(* Logix 5000 project; controller R5_CSS vendor 1 type 14 code 74 rev 19.11; software revision 19.01; part 6 of 18 *)
(* tags used below, declared in another part *)
   AC102A : ANALYTICAL;   // QUENCH WATER CONDUCTIVITY CONTROL
   AlarmMaster : DINT;
   AlarmMasterDisable : BOOL;
   AlarmMasterResetTON : TIMER;
   AlarmResetPB : BOOL;
   FC101 : FLOW_CONTROL;   // QUENCH BASIN FLOW TRANSMITTER CONTROL
   FC108 : FLOW_CONTROL;   // QUENCH FEED FLOW TRANSMITTER
   FC140A : FLOW_CONTROL;   // QUENCH TOWER UPPER SPRAY FLOW CONTROL
   FC140B : FLOW_CONTROL;   // QUENCH TOWER LOWER SPRAY FLOW CONTROL
   FC365 : FLOW_CONTROL;   // COALESCER PROCESS IMPURITY FLOW CONTROL
   FireFlowAlarmFromUTL : BOOL;
   HMI_ShowReboot : BOOL;
   HMI_ShowRebootTmr : TIMER;
   Instrument_LOS : BOOL[32];
   LC205 : LEVEL_CONTROL;   // OVERHEAD CONDENSER BASIN LEVEL CONTROL
   LC302 : LEVEL_CONTROL;   // COALESCER OIL CHAMBER LEVEL CONTROL
   LC303A : LEVEL_CONTROL;   // AQUEOUS PHASE OF PRIMARY SETTLER
   Option_F1_Occupancy : BOOL;   // STATUS FROM UTL PLC 0=DISABLED 1=ENABLED
   P101_OK_TON : TIMER;
   P101A_OK : BOOL;
   P101B_OK : BOOL;
   P302A : PUMP_CONTROL;
   P302B : PUMP_CONTROL;
   P303_OK_TON : TIMER;
   P303A_OK : BOOL;
   P303B_OK : BOOL;
   PC101A : PRESSURE_CONTROL;   // LOWER QUENCH TOWER PRESSURE TRANSMITTER
   PC101B : PRESSURE_CONTROL;   // UPPER QUENCH TOWER PRESSURE TRANSMITTER PRESSURE CONTOL
   PC407B : PRESSURE_CONTROL;   // POST HX LOW PRESSURE TRANSMITTER
   TC101A : TEMP_CONTROL;   // QUENCH BASIN TRANSFER BASIN A TEMPERATURE CONTROL
   TC108 : TEMP_CONTROL;   // QUENCH TOWER EXIT GAS TEMPERATURE CONTROL
   TC114A : TEMP_CONTROL;   // QUENCH BASIN SHELL TEMPERATURE CONTROL
   TMR_FAULT : DINT;
   UTL_Comms : DINT[3];
   UTL_CommsLossAlm : BOOL;
(* MainProgram, continued *)

ROUTINE A4_Alarms_General   (* ladder *)
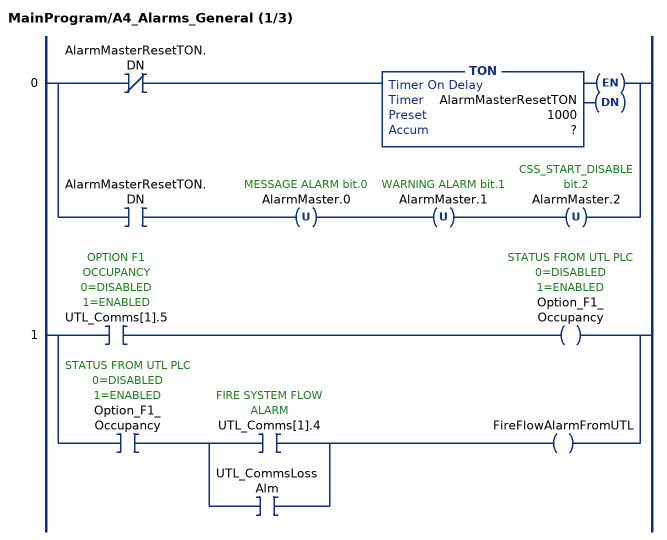
   0: [XIO(AlarmMasterResetTON.DN) TON(AlarmMasterResetTON,?,?) ,XIC(AlarmMasterResetTON.DN) OTU(AlarmMaster.0) OTU(AlarmMaster.1) OTU(AlarmMaster.2) ];
   1: [XIC(UTL_Comms[1].5) OTE(Option_F1_Occupancy) ,XIC(Option_F1_Occupancy) [XIC(UTL_Comms[1].4) ,XIC(UTL_CommsLossAlm) ] OTE(FireFlowAlarmFromUTL) ];
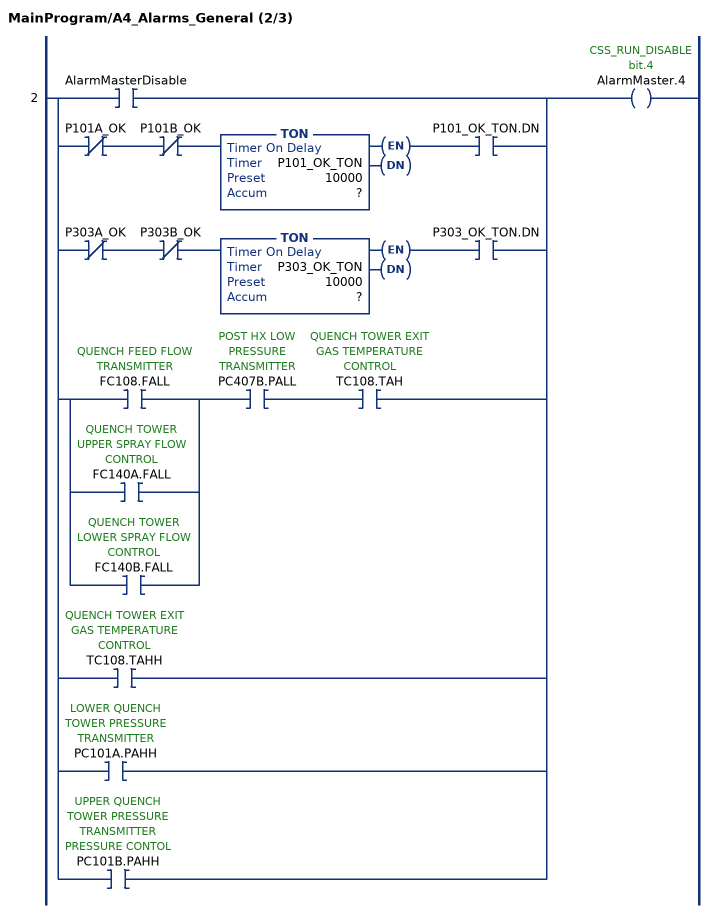
   2: [XIC(AlarmMasterDisable) ,XIO(P101A_OK) XIO(P101B_OK) TON(P101_OK_TON,?,?) XIC(P101_OK_TON.DN) ,XIO(P303A_OK) XIO(P303B_OK) TON(P303_OK_TON,?,?) XIC(P303_OK_TON.DN) ,[XIC(FC108.FALL) ,XIC(FC140A.FALL) ,XIC(FC140B.FALL) ] XIC(PC407B.PALL) XIC(TC108.TAH) ,XIC(TC108.TAHH) ,XIC(PC101A.PAHH) ,XIC(PC101B.PAHH) ]OTE(AlarmMaster.4);
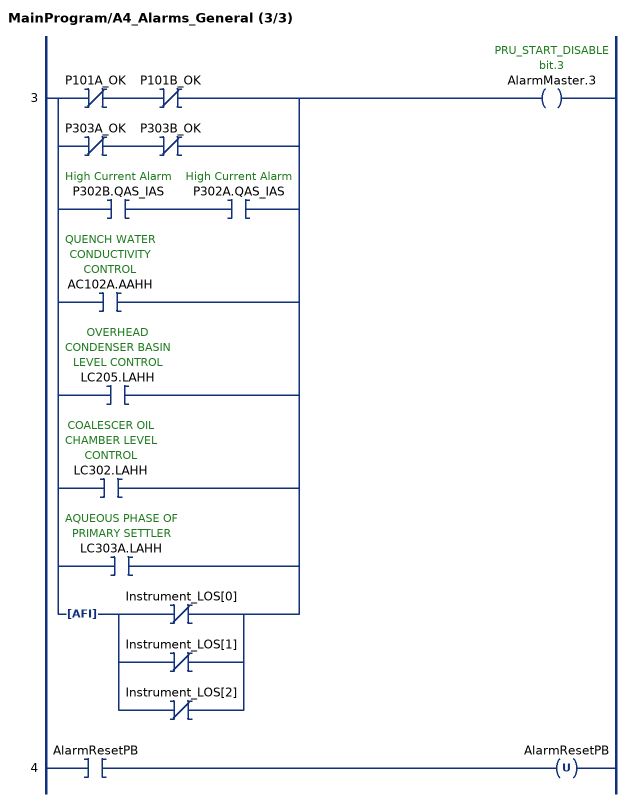
   3: [XIO(P101A_OK) XIO(P101B_OK) ,XIO(P303A_OK) XIO(P303B_OK) ,XIC(P302B.QAS_IAS) XIC(P302A.QAS_IAS) ,XIC(AC102A.AAHH) ,XIC(LC205.LAHH) ,XIC(LC302.LAHH) ,XIC(LC303A.LAHH) ,AFI() [XIO(Instrument_LOS[0]) ,XIO(Instrument_LOS[1]) ,XIO(Instrument_LOS[2]) ] ]OTE(AlarmMaster.3);
   4: XIC(AlarmResetPB)OTU(AlarmResetPB);
END_ROUTINE

ROUTINE A5a_LOAD_START_UP_PARAMETERS   (* ladder *)
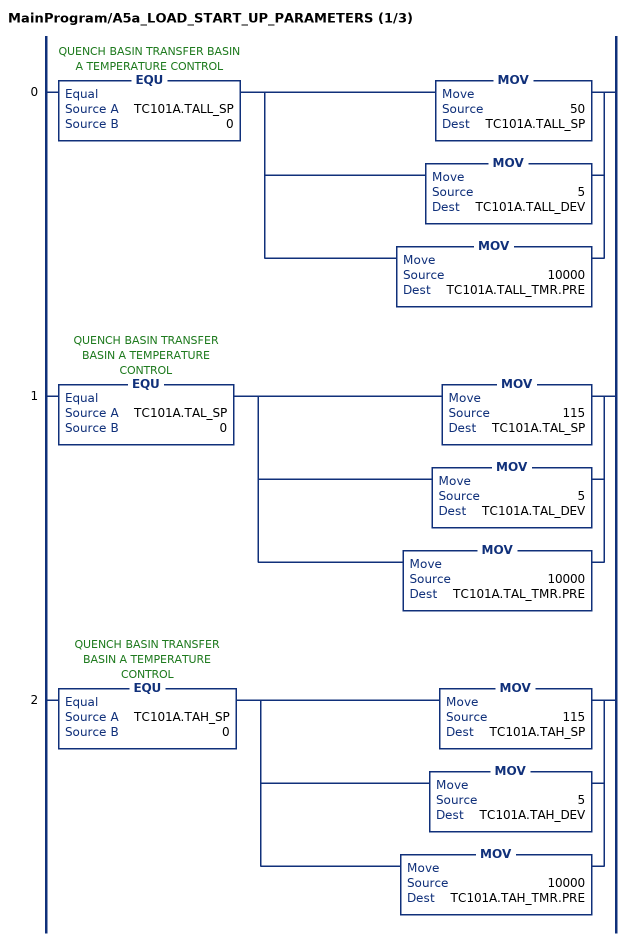
   0: EQU(TC101A.TALL_SP,0)[MOV(50,TC101A.TALL_SP) ,MOV(5,TC101A.TALL_DEV) ,MOV(10000,TC101A.TALL_TMR.PRE) ];
   1: EQU(TC101A.TAL_SP,0)[MOV(115,TC101A.TAL_SP) ,MOV(5,TC101A.TAL_DEV) ,MOV(10000,TC101A.TAL_TMR.PRE) ];
   2: EQU(TC101A.TAH_SP,0)[MOV(115,TC101A.TAH_SP) ,MOV(5,TC101A.TAH_DEV) ,MOV(10000,TC101A.TAH_TMR.PRE) ];
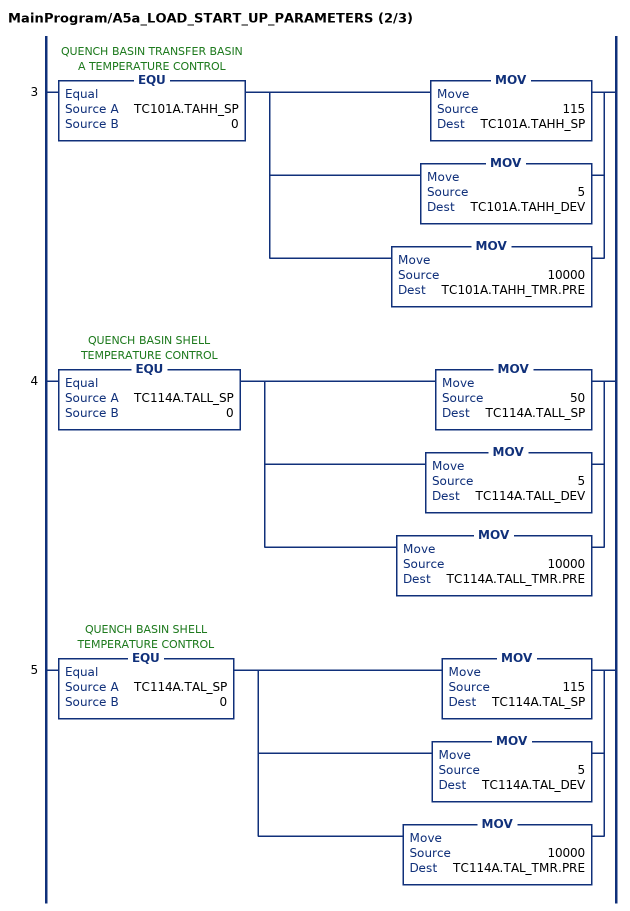
   3: EQU(TC101A.TAHH_SP,0)[MOV(115,TC101A.TAHH_SP) ,MOV(5,TC101A.TAHH_DEV) ,MOV(10000,TC101A.TAHH_TMR.PRE) ];
   4: EQU(TC114A.TALL_SP,0)[MOV(50,TC114A.TALL_SP) ,MOV(5,TC114A.TALL_DEV) ,MOV(10000,TC114A.TALL_TMR.PRE) ];
   5: EQU(TC114A.TAL_SP,0)[MOV(115,TC114A.TAL_SP) ,MOV(5,TC114A.TAL_DEV) ,MOV(10000,TC114A.TAL_TMR.PRE) ];
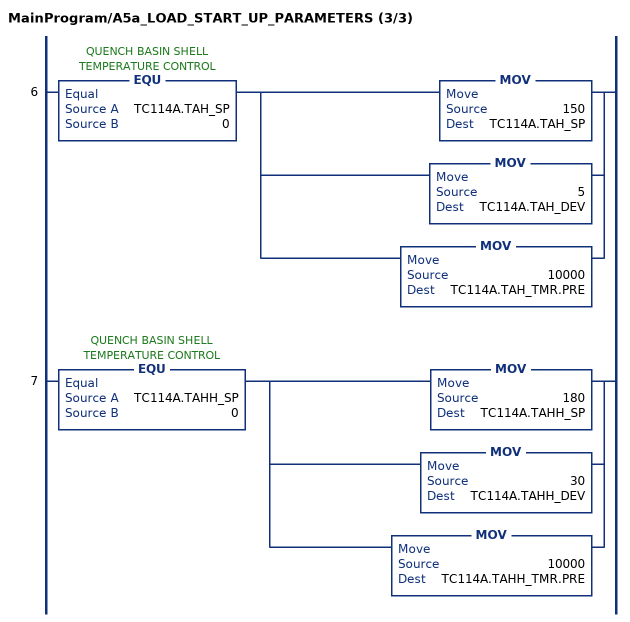
   6: EQU(TC114A.TAH_SP,0)[MOV(150,TC114A.TAH_SP) ,MOV(5,TC114A.TAH_DEV) ,MOV(10000,TC114A.TAH_TMR.PRE) ];
   7: EQU(TC114A.TAHH_SP,0)[MOV(180,TC114A.TAHH_SP) ,MOV(30,TC114A.TAHH_DEV) ,MOV(10000,TC114A.TAHH_TMR.PRE) ];
END_ROUTINE

ROUTINE A5b_LOCAL_HMI   (* ladder *)
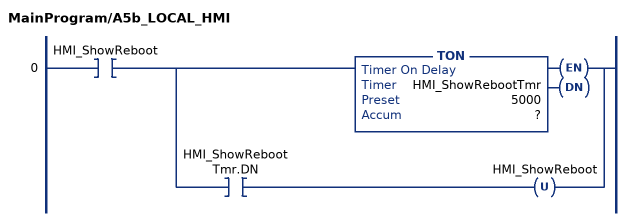
   0: XIC(HMI_ShowReboot)[TON(HMI_ShowRebootTmr,?,?) ,XIC(HMI_ShowRebootTmr.DN) OTU(HMI_ShowReboot) ];
END_ROUTINE

ROUTINE AT102A_QuenchWaterConductivity   (* ladder *)
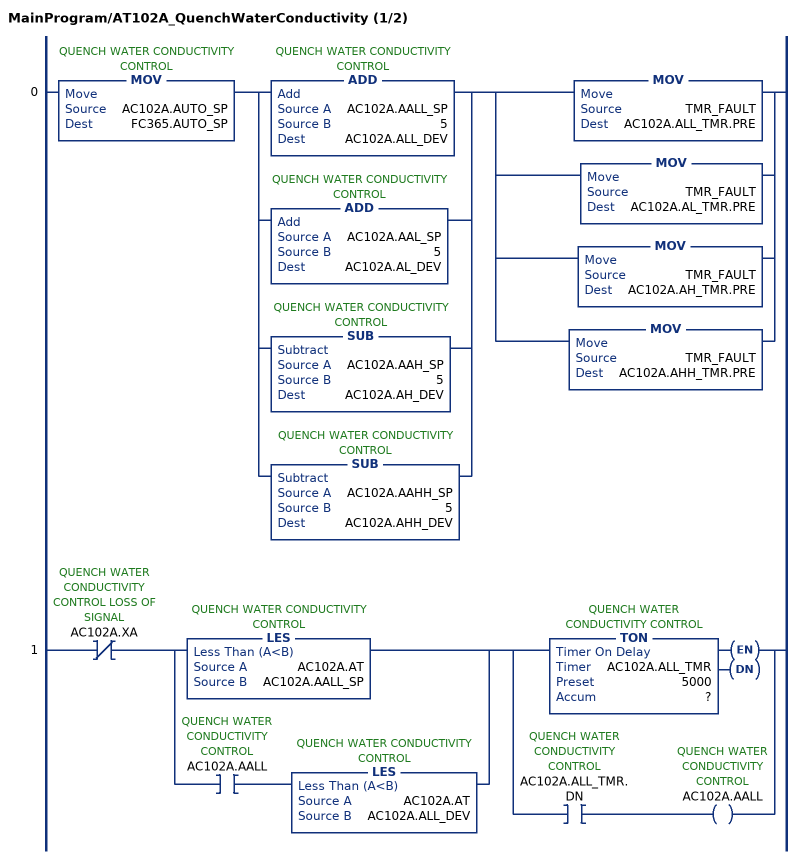
   0: MOV(AC102A.AUTO_SP,FC365.AUTO_SP)[ADD(AC102A.AALL_SP,5,AC102A.ALL_DEV) ,ADD(AC102A.AAL_SP,5,AC102A.AL_DEV) ,SUB(AC102A.AAH_SP,5,AC102A.AH_DEV) ,SUB(AC102A.AAHH_SP,5,AC102A.AHH_DEV) ][MOV(TMR_FAULT,AC102A.ALL_TMR.PRE) ,MOV(TMR_FAULT,AC102A.AL_TMR.PRE) ,MOV(TMR_FAULT,AC102A.AH_TMR.PRE) ,MOV(TMR_FAULT,AC102A.AHH_TMR.PRE) ];
   1: XIO(AC102A.XA)[LES(AC102A.AT,AC102A.AALL_SP) ,XIC(AC102A.AALL) LES(AC102A.AT,AC102A.ALL_DEV) ][TON(AC102A.ALL_TMR,?,?) ,XIC(AC102A.ALL_TMR.DN) OTE(AC102A.AALL) ];
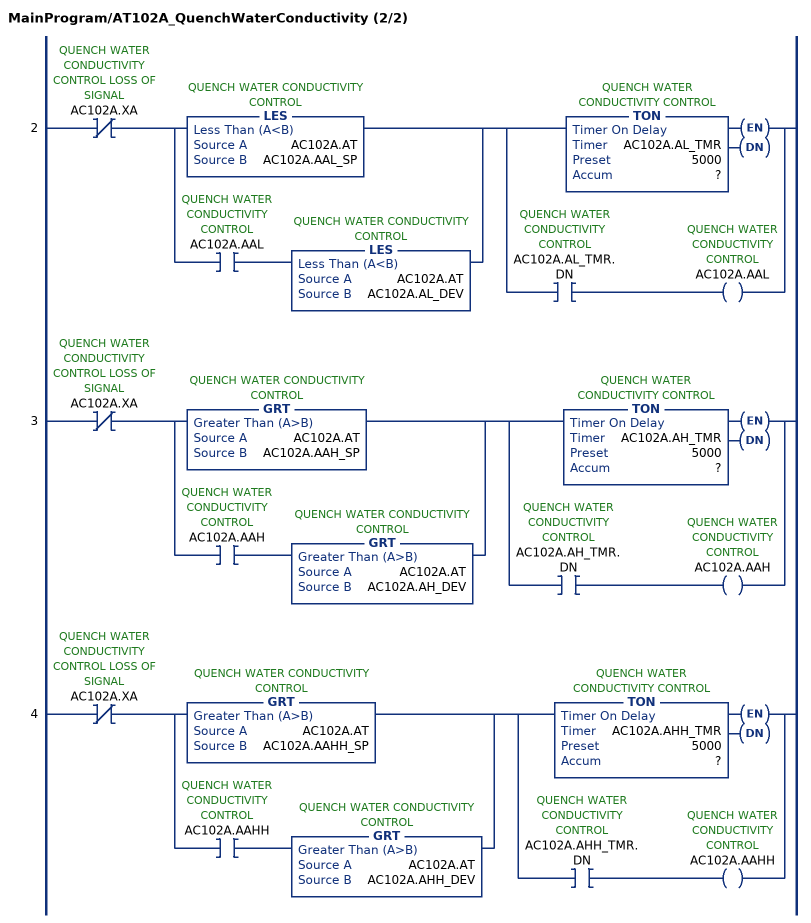
   2: XIO(AC102A.XA)[LES(AC102A.AT,AC102A.AAL_SP) ,XIC(AC102A.AAL) LES(AC102A.AT,AC102A.AL_DEV) ][TON(AC102A.AL_TMR,?,?) ,XIC(AC102A.AL_TMR.DN) OTE(AC102A.AAL) ];
   3: XIO(AC102A.XA)[GRT(AC102A.AT,AC102A.AAH_SP) ,XIC(AC102A.AAH) GRT(AC102A.AT,AC102A.AH_DEV) ][TON(AC102A.AH_TMR,?,?) ,XIC(AC102A.AH_TMR.DN) OTE(AC102A.AAH) ];
   4: XIO(AC102A.XA)[GRT(AC102A.AT,AC102A.AAHH_SP) ,XIC(AC102A.AAHH) GRT(AC102A.AT,AC102A.AHH_DEV) ][TON(AC102A.AHH_TMR,?,?) ,XIC(AC102A.AHH_TMR.DN) OTE(AC102A.AAHH) ];
END_ROUTINE

ROUTINE FC101_BasinFlow   (* ladder *)
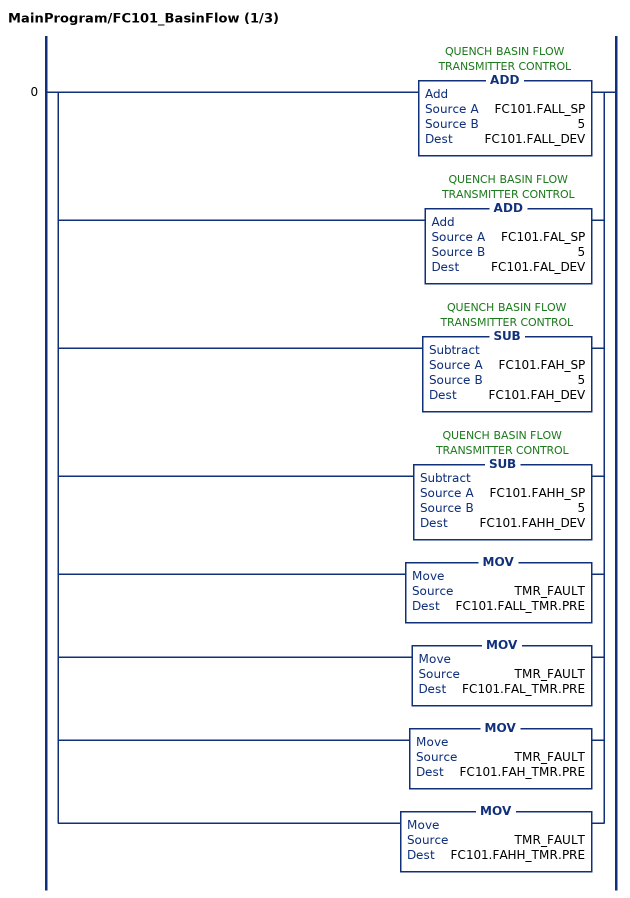
   0: [ADD(FC101.FALL_SP,5,FC101.FALL_DEV) ,ADD(FC101.FAL_SP,5,FC101.FAL_DEV) ,SUB(FC101.FAH_SP,5,FC101.FAH_DEV) ,SUB(FC101.FAHH_SP,5,FC101.FAHH_DEV) ,MOV(TMR_FAULT,FC101.FALL_TMR.PRE) ,MOV(TMR_FAULT,FC101.FAL_TMR.PRE) ,MOV(TMR_FAULT,FC101.FAH_TMR.PRE) ,MOV(TMR_FAULT,FC101.FAHH_TMR.PRE) ];
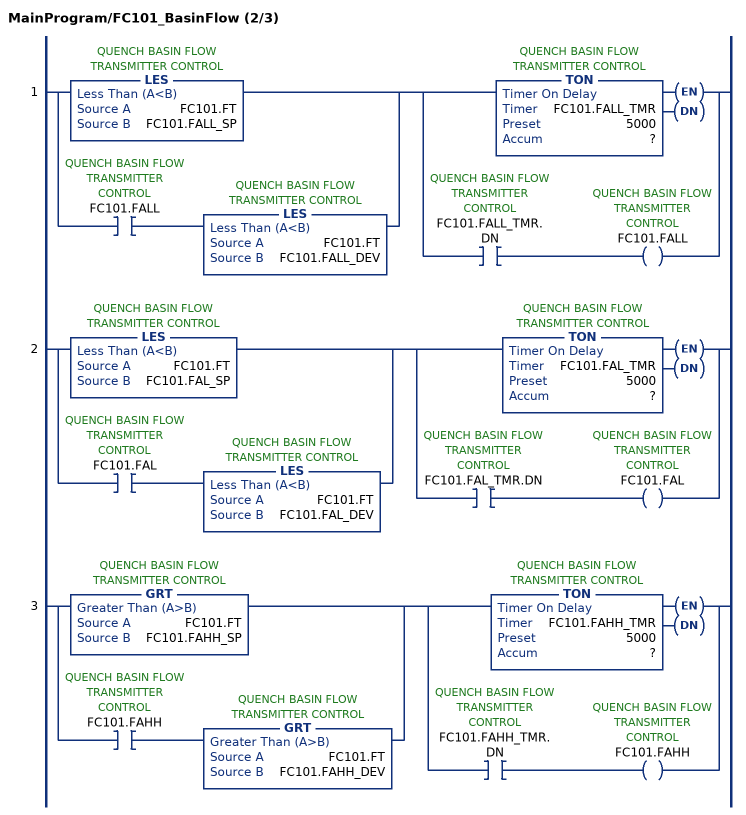
   1: [LES(FC101.FT,FC101.FALL_SP) ,XIC(FC101.FALL) LES(FC101.FT,FC101.FALL_DEV) ][TON(FC101.FALL_TMR,?,?) ,XIC(FC101.FALL_TMR.DN) OTE(FC101.FALL) ];
   2: [LES(FC101.FT,FC101.FAL_SP) ,XIC(FC101.FAL) LES(FC101.FT,FC101.FAL_DEV) ][TON(FC101.FAL_TMR,?,?) ,XIC(FC101.FAL_TMR.DN) OTE(FC101.FAL) ];
   3: [GRT(FC101.FT,FC101.FAHH_SP) ,XIC(FC101.FAHH) GRT(FC101.FT,FC101.FAHH_DEV) ][TON(FC101.FAHH_TMR,?,?) ,XIC(FC101.FAHH_TMR.DN) OTE(FC101.FAHH) ];
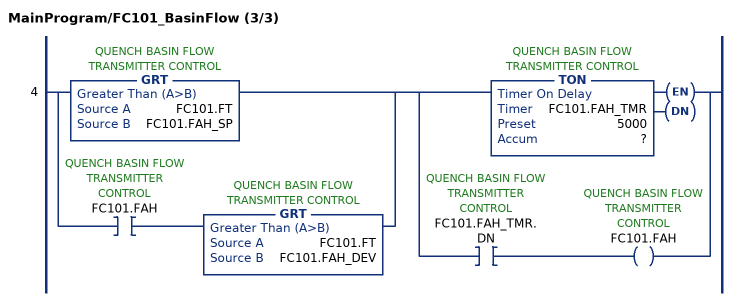
   4: [GRT(FC101.FT,FC101.FAH_SP) ,XIC(FC101.FAH) GRT(FC101.FT,FC101.FAH_DEV) ][TON(FC101.FAH_TMR,?,?) ,XIC(FC101.FAH_TMR.DN) OTE(FC101.FAH) ];
END_ROUTINE

ROUTINE FC108_QuenchTowerFlow   (* ladder *)
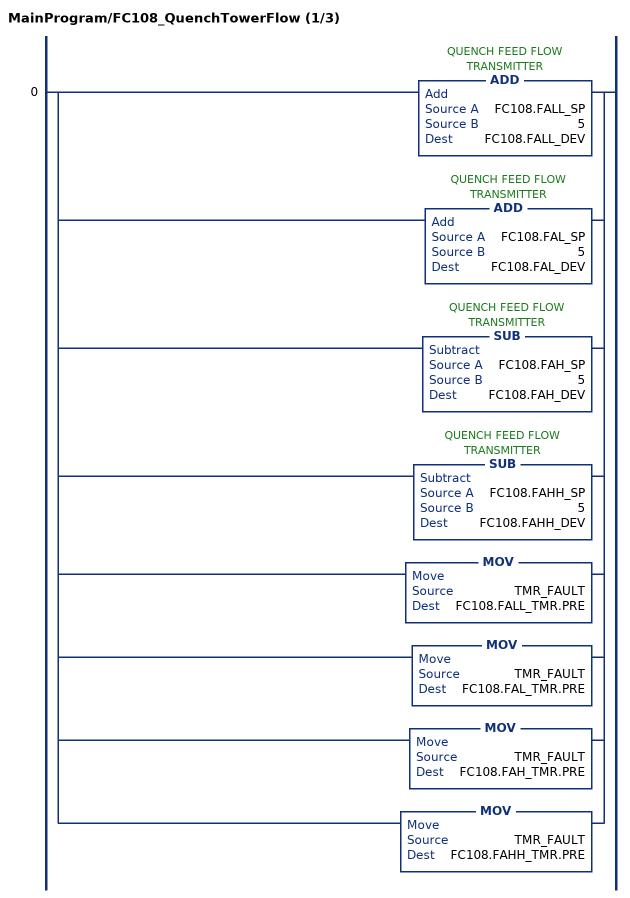
   0: [ADD(FC108.FALL_SP,5,FC108.FALL_DEV) ,ADD(FC108.FAL_SP,5,FC108.FAL_DEV) ,SUB(FC108.FAH_SP,5,FC108.FAH_DEV) ,SUB(FC108.FAHH_SP,5,FC108.FAHH_DEV) ,MOV(TMR_FAULT,FC108.FALL_TMR.PRE) ,MOV(TMR_FAULT,FC108.FAL_TMR.PRE) ,MOV(TMR_FAULT,FC108.FAH_TMR.PRE) ,MOV(TMR_FAULT,FC108.FAHH_TMR.PRE) ];
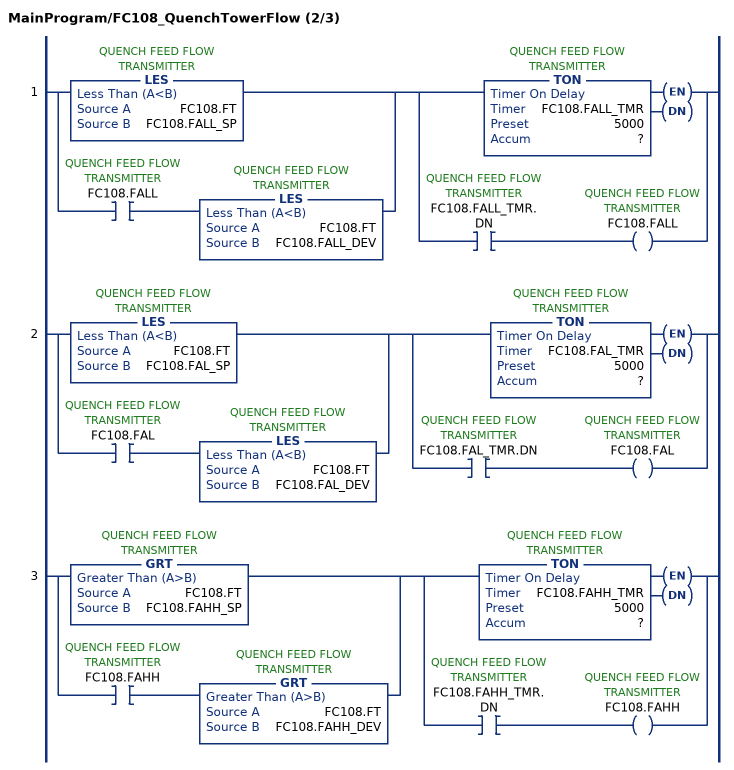
   1: [LES(FC108.FT,FC108.FALL_SP) ,XIC(FC108.FALL) LES(FC108.FT,FC108.FALL_DEV) ][TON(FC108.FALL_TMR,?,?) ,XIC(FC108.FALL_TMR.DN) OTE(FC108.FALL) ];
   2: [LES(FC108.FT,FC108.FAL_SP) ,XIC(FC108.FAL) LES(FC108.FT,FC108.FAL_DEV) ][TON(FC108.FAL_TMR,?,?) ,XIC(FC108.FAL_TMR.DN) OTE(FC108.FAL) ];
   3: [GRT(FC108.FT,FC108.FAHH_SP) ,XIC(FC108.FAHH) GRT(FC108.FT,FC108.FAHH_DEV) ][TON(FC108.FAHH_TMR,?,?) ,XIC(FC108.FAHH_TMR.DN) OTE(FC108.FAHH) ];
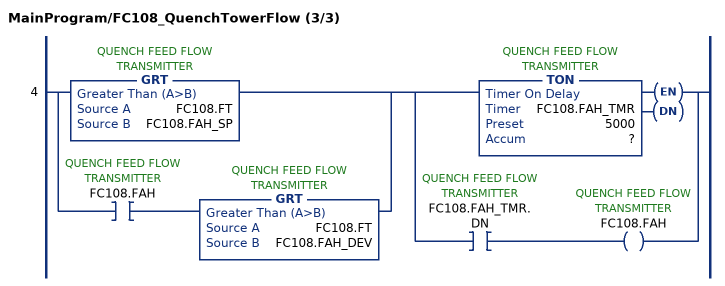
   4: [GRT(FC108.FT,FC108.FAH_SP) ,XIC(FC108.FAH) GRT(FC108.FT,FC108.FAH_DEV) ][TON(FC108.FAH_TMR,?,?) ,XIC(FC108.FAH_TMR.DN) OTE(FC108.FAH) ];
END_ROUTINE

ROUTINE FC140A_QuenchWaterUpperSprayFlow   (* ladder *)
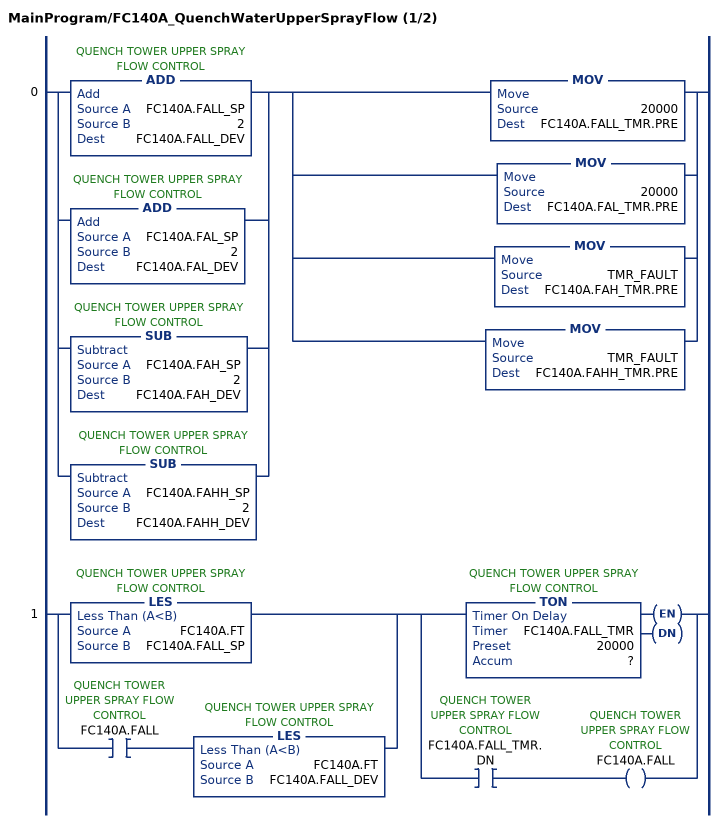
   0: [ADD(FC140A.FALL_SP,2,FC140A.FALL_DEV) ,ADD(FC140A.FAL_SP,2,FC140A.FAL_DEV) ,SUB(FC140A.FAH_SP,2,FC140A.FAH_DEV) ,SUB(FC140A.FAHH_SP,2,FC140A.FAHH_DEV) ][MOV(20000,FC140A.FALL_TMR.PRE) ,MOV(20000,FC140A.FAL_TMR.PRE) ,MOV(TMR_FAULT,FC140A.FAH_TMR.PRE) ,MOV(TMR_FAULT,FC140A.FAHH_TMR.PRE) ];
   1: [LES(FC140A.FT,FC140A.FALL_SP) ,XIC(FC140A.FALL) LES(FC140A.FT,FC140A.FALL_DEV) ][TON(FC140A.FALL_TMR,?,?) ,XIC(FC140A.FALL_TMR.DN) OTE(FC140A.FALL) ];
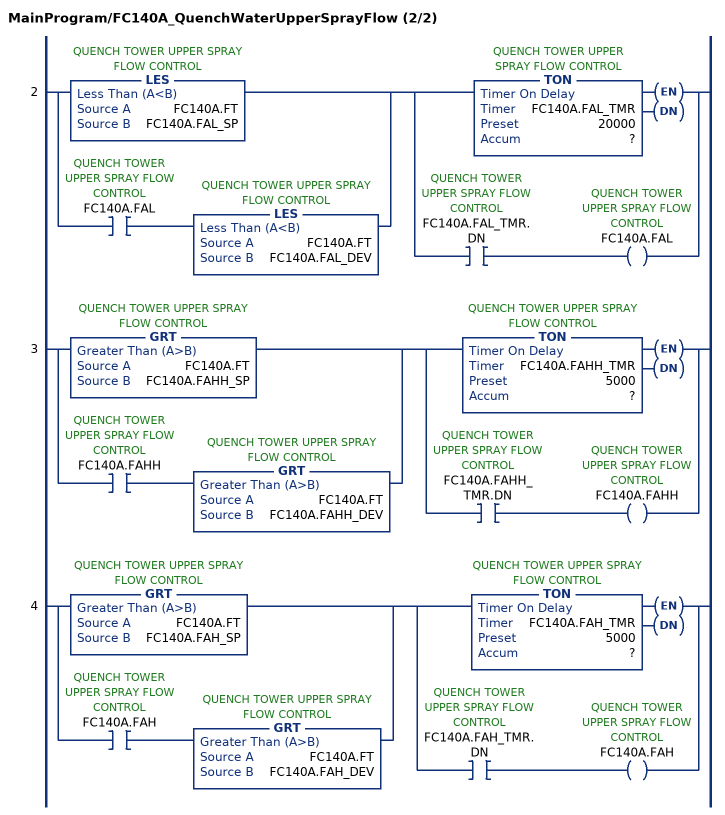
   2: [LES(FC140A.FT,FC140A.FAL_SP) ,XIC(FC140A.FAL) LES(FC140A.FT,FC140A.FAL_DEV) ][TON(FC140A.FAL_TMR,?,?) ,XIC(FC140A.FAL_TMR.DN) OTE(FC140A.FAL) ];
   3: [GRT(FC140A.FT,FC140A.FAHH_SP) ,XIC(FC140A.FAHH) GRT(FC140A.FT,FC140A.FAHH_DEV) ][TON(FC140A.FAHH_TMR,?,?) ,XIC(FC140A.FAHH_TMR.DN) OTE(FC140A.FAHH) ];
   4: [GRT(FC140A.FT,FC140A.FAH_SP) ,XIC(FC140A.FAH) GRT(FC140A.FT,FC140A.FAH_DEV) ][TON(FC140A.FAH_TMR,?,?) ,XIC(FC140A.FAH_TMR.DN) OTE(FC140A.FAH) ];
END_ROUTINE

ROUTINE FC140B_QuenchWaterLowerSprayFlow   (* ladder *)
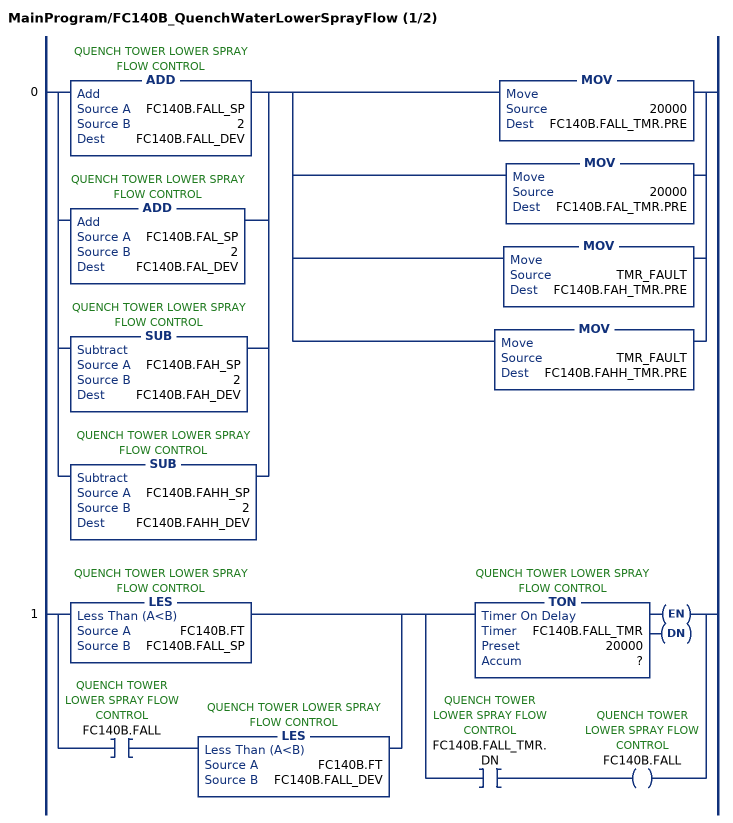
   0: [ADD(FC140B.FALL_SP,2,FC140B.FALL_DEV) ,ADD(FC140B.FAL_SP,2,FC140B.FAL_DEV) ,SUB(FC140B.FAH_SP,2,FC140B.FAH_DEV) ,SUB(FC140B.FAHH_SP,2,FC140B.FAHH_DEV) ][MOV(20000,FC140B.FALL_TMR.PRE) ,MOV(20000,FC140B.FAL_TMR.PRE) ,MOV(TMR_FAULT,FC140B.FAH_TMR.PRE) ,MOV(TMR_FAULT,FC140B.FAHH_TMR.PRE) ];
   1: [LES(FC140B.FT,FC140B.FALL_SP) ,XIC(FC140B.FALL) LES(FC140B.FT,FC140B.FALL_DEV) ][TON(FC140B.FALL_TMR,?,?) ,XIC(FC140B.FALL_TMR.DN) OTE(FC140B.FALL) ];
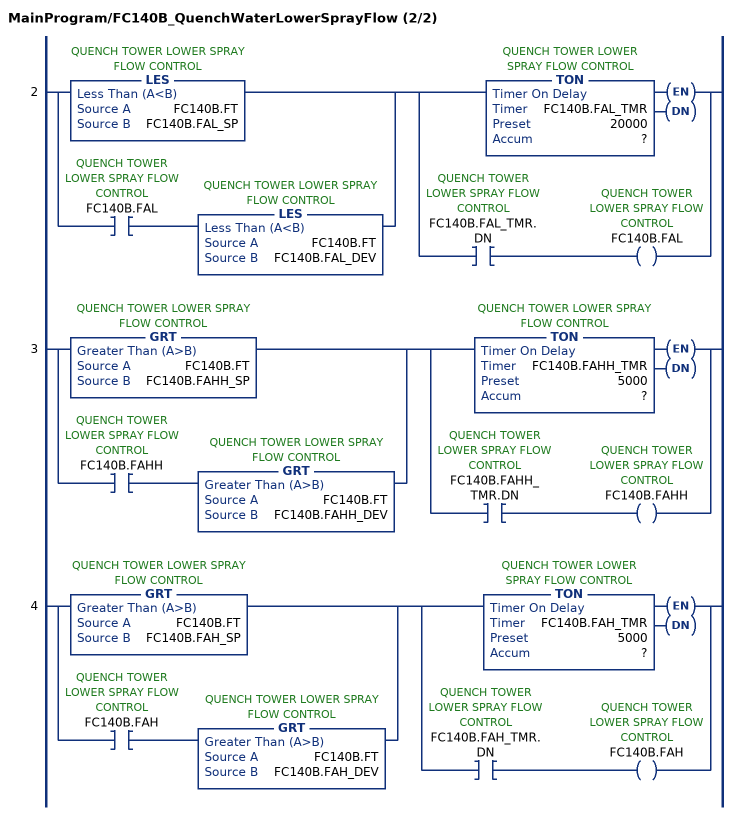
   2: [LES(FC140B.FT,FC140B.FAL_SP) ,XIC(FC140B.FAL) LES(FC140B.FT,FC140B.FAL_DEV) ][TON(FC140B.FAL_TMR,?,?) ,XIC(FC140B.FAL_TMR.DN) OTE(FC140B.FAL) ];
   3: [GRT(FC140B.FT,FC140B.FAHH_SP) ,XIC(FC140B.FAHH) GRT(FC140B.FT,FC140B.FAHH_DEV) ][TON(FC140B.FAHH_TMR,?,?) ,XIC(FC140B.FAHH_TMR.DN) OTE(FC140B.FAHH) ];
   4: [GRT(FC140B.FT,FC140B.FAH_SP) ,XIC(FC140B.FAH) GRT(FC140B.FT,FC140B.FAH_DEV) ][TON(FC140B.FAH_TMR,?,?) ,XIC(FC140B.FAH_TMR.DN) OTE(FC140B.FAH) ];
END_ROUTINE
